(* CoDeSys 2.3 export: ACTUATORS.EXP *)

(* POU ACTUATORS, FBD *)
FUNCTION_BLOCK ACTUATORS
VAR_INPUT
	iSTATE		:	INT;
END_VAR
VAR_OUTPUT
	_xROTARY_MOTOR		:	BOOL;
	_xPUNCH					:	BOOL;
	_xLOWER_DRILL			:	BOOL;
	_xRAISE_DRILL			:	BOOL;
	_xDRILL					:	BOOL;
	_xDRILL_PUNCH			:	BOOL;
END_VAR
VAR
END_VAR
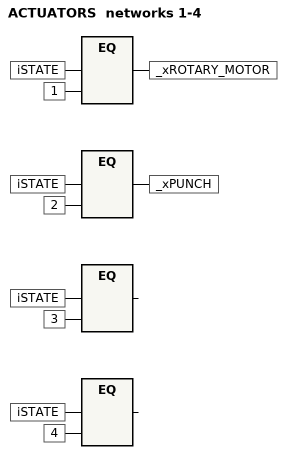
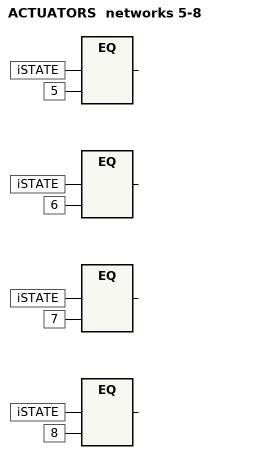
_FBD_ (* Function Block Diagram *)
NETWORK 1
	EQ(iSTATE, 1) => _xROTARY_MOTOR
NETWORK 2
	EQ(iSTATE, 2) => _xPUNCH
NETWORK 3
	EQ(iSTATE, 3)
NETWORK 4
	EQ(iSTATE, 4)
NETWORK 5
	EQ(iSTATE, 5)
NETWORK 6
	EQ(iSTATE, 6)
NETWORK 7
	EQ(iSTATE, 7)
NETWORK 8
	EQ(iSTATE, 8)
_END_FBD_
(* the same logic as Structured Text *)
(* Network 1 *)
_xROTARY_MOTOR := iSTATE = 1;
(* Network 2 *)
_xPUNCH := iSTATE = 2;
(* Network 3: see the listing above *)
(* Network 4: see the listing above *)
(* Network 5: see the listing above *)
(* Network 6: see the listing above *)
(* Network 7: see the listing above *)
(* Network 8: see the listing above *)
END_FUNCTION_BLOCK
